(*
Nazwa:			FB_MoveRegister
Opis:			Blok przesuniecia rejestru formatek
Wersja:			v0.3 		
Data:			2018-11-16
Autor:			DP
Urzadzenia:		 
Konfiguracja:	
Info:
- Są dwa rejestry, wejściowy i wyjsciowy (struktury)
- Jezeli rejestr ma np. 6 elementów to za kazdym razem po wykryciu trigera program będzie
	1 wejściowy przesuwał na 1 wolny (nie ma formatki) wyjściowy
	kasował 1 rejestr wejściowy
	przesuwal rejetr wejsciowy 2 na 1(przeniesiony i skasowany), 3 na 2, 4 na 3, 5 na 4, 6 na 5 i kasowal 6wejsciowy
	tym sposobem po 6 trigerach caly rejestr wejsciowy powinien być na wyjsciowym
	np po 3 trigerach na wyjsciowym powinny byc zajete 1 do 3 i na wejsciowym 1 do 3
Błędy:
1 - nie wyszło z pętli for
2 - formatka już jest w rejestrze
Uwagi:
- 
Zmiany:
2018-09-18 Dodano sprawdzanie nasadek
2018-06-14 DP Pierwsza wersja
*)

FUNCTION_BLOCK FB_MoveRegisterLF
VAR_INPUT
	bFirstCycle:BOOL;					//Pierwszy cykl, zeby na początku nie wykrywało zbocza opadającego
	bTrigger :BOOL;						// Przesuniecie tablicy o jeden
	tTriggerFilterTimeOn:TIME:=T#0MS;	// Czas filtrowania wejścia Trigger na załączenie
	tTriggerFilterTimeOff:TIME:=T#0MS;	// Czas filtrowania wejścia Trigger na wyłączenie
	bTriggerBottle :BOOL;				// Zapisywanie czy jest butelka czy nie (jezeli kontrola wlączona)
	bWithBottleControl: BOOL;			// Włączona opcja kontroli butelek
	bWithCapControl:BOOL;				// Wlaczona kontrola nasadek
	bWithFormControlTrigerCounter:BOOL;	// Jezeku na trigercontrol nie ma formatki do przesunięcia to stwórz nową
	bMoveOnlyToLastExitRegister:BOOL;	// Przepisuj rejestr wejściowy tylko na ostatni wyjściowy bez przesunięcia wyjściowego
	bMoveOnlyIfFormPresent:BOOL;		// Przepisuj tylko jak jest formatka
	bRotateEntranceRegisterBefore:BOOL;	// Najpierw przesuń rejestr wejściowy a następnie z niego zabierz
	bNoKeepTryingMove:BOOL;				// Dalej przepisuj jezeli nie ma miejsca
	bTriggerCap: BOOL;					// Truger wykrycia nasadki
	bReset :BOOL;						// Czyszczenie tablic
	iEntranceArrayElements :UINT; 		// Wartość koncowa tablicy
	iExitArrayElements :UINT; 			// Wartość koncowa tablicy
	bInvertWriting :BOOL;				// Wpisywanie odwrotne zamist z 1entrance na 1exit to 1entrance na 6exit	
	eClearPackageState :S_PackageState; // Czysty rejestr
END_VAR
VAR_IN_OUT
	bTriggerCounter :BOOL;		// Triger ktory jest kasowany
	eEntranceState :ARRAY [1..17] OF S_PackageState;	
	eExitState :ARRAY [1..17] OF S_PackageState;
	bKeepTryingMove :BOOL;		// Probuj dalej zapisać formatki aż się któraś zwolni
END_VAR

VAR_OUTPUT	
	bError :BOOL; 				// Błąd
	iError: UINT;				// Nr Błędu
	bTriggerDone :BOOL; 		// Wykonano przesunięcie
	bTriggerFilteredOUT:BOOL;	//Wyjscie przefiltrowanego sygnalu wejsciowego
END_VAR

VAR
	i:UINT;						// Zmienna w tablicy
	k:UINT;						// Pomocnicza zmienna do zapisywnia czy jest butelka
	rtbTrigger :R_TRIG;			// Reaguje na zbocze
	rtbTriggerBottle :R_TRIG;	// Reaguje na zbocze
	rtbReset :R_TRIG;			// Reaguje na zbocze
	TimerResetErrors :TON;		// Reset Błedu
	nFormCounter :UINT;					//Licznik formatek
	r1,r2:UINT;
	bBottlePresent: BOOL;				//Zmienna pomocnicza ze wykryto butelkę
	bCapPresent: BOOL;					//Zmienna pomocnicza ze wykryto butelkę
	j: UINT;
	tonTriggerFilterTimeOn: TON;
	bTriggerFiltered: BOOL;
	tofTriggerFilterTimeOff: TOF;
	tonTriggerFilterTimeBeforeTrigger: TON;
END_VAR

//Filtrowanie sygnału wejściowego
tofTriggerFilterTimeOff	(IN:=bTrigger, PT:=tTriggerFilterTimeOff);
tonTriggerFilterTimeOn	(IN:=tofTriggerFilterTimeOff.Q, PT:=tTriggerFilterTimeOn);
bTriggerFiltered 		:= tonTriggerFilterTimeOn.Q;
bTriggerFilteredOUT		:= bTriggerFiltered ;

//TRIGI I TIMERY
IF bWithBottleControl THEN
	rtbTrigger 	(CLK := NOT bTriggerFiltered, Q=>);
	rtbTriggerBottle 	(CLK := NOT bTriggerBottle, Q=>);
ELSIF bWithCapControl THEN
	rtbTrigger 	(CLK := NOT bTriggerFiltered, Q=>);
ELSE
	rtbTrigger 	(CLK := bTriggerFiltered, Q=>);
	rtbTriggerBottle 	(CLK := bTriggerBottle, Q=>);
END_IF

rtbReset 	(CLK := bReset, Q=>);
TimerResetErrors (IN:= bError, PT:=T#1000MS, Q=>);

//RESETOWANIE BLEDU
IF TimerResetErrors.Q THEN
	bError := FALSE;
END_IF

//KASOWANIE ZMIENNYCH
bTriggerDone := FALSE;

//JEZELI WLACZONO KONTROLE BUTELEK TO NADPISUJ REJESTR CZY JEST BUTELKA
IF bWithBottleControl AND bTrigger AND bTriggerBottle AND NOT bKeepTryingMove THEN //Jezeli od wykrycia formatki liczy TIMER i wykryło butelke to wpisz do rejestru że jest butelka
	eEntranceState[1].bBottlePresent := TRUE;
	eEntranceState[1].bFormPresent := TRUE;
	bBottlePresent := TRUE; // Wpisuje że jest butelka jezeli wystąpi sygnał podczas trwania czujnika formatki
ELSIF bWithBottleControl AND rtbTrigger.Q AND NOT bBottlePresent AND  NOT bKeepTryingMove AND bFirstCycle THEN
	eEntranceState[1].bBottlePresent := FALSE;
	eEntranceState[1].bFormPresent := TRUE; // jeżeli zanik czujnik formatki i nie było formatki to wpisz ze nie było butelki
END_IF
//JEZELI WLACZONO KONTROLE NASADEk TO NADPISUJ REJESTR CZY JEST BUTELKA 
(*IF bWithCapControl AND bTrigger AND bTriggerCap AND NOT bKeepTryingMove THEN //Jezeli od wykrycia formatki liczy TIMER i wykryło butelke to wpisz do rejestru że jest butelka
	eEntranceState[1].bCapPutted := TRUE;
	eEntranceState[1].bCapOK := TRUE; eEntranceState[1].bBottlePresent:= TRUE;//Zmiana nowa
	eEntranceState[1].bFormPresent := TRUE;
	bCapPresent := TRUE; // Wpisuje że jest butelka jezeli wystąpi sygnał podczas trwania czujnika formatki*)
	//ZMIANA LU 192
IF bWithCapControl AND bTriggerCap AND NOT bKeepTryingMove THEN //Jezeli od wykrycia formatki liczy TIMER i wykryło butelke to wpisz do rejestru że jest butelka
	eEntranceState[1].bCapPutted := TRUE;
	eEntranceState[1].bCapOK := TRUE; eEntranceState[1].bBottlePresent:= TRUE;//Zmiana nowa
	eEntranceState[1].bFormPresent := TRUE;
	bCapPresent := TRUE; // Wpisuje że jest butelka jezeli wystąpi sygnał podczas trwania czujnika formatki	
ELSIF bWithCapControl AND rtbTrigger.Q AND NOT bCapPresent AND  NOT bKeepTryingMove AND bFirstCycle THEN
	eEntranceState[1].bCapPutted := TRUE;
	eEntranceState[1].bCapOK:= FALSE;
	eEntranceState[1].bFormPresent := TRUE; // jeżeli zanik czujnik formatki i nie było formatki to wpisz ze nie było butelki
END_IF
//JEZELI WLACZONO SPRAWDZANIE FORMATEK Z TRIGERCOUNTER TO
IF bWithFormControlTrigerCounter  AND (bTriggerCounter OR rtbTrigger.Q) AND NOT bKeepTryingMove AND bFirstCycle THEN //Zmiena UBL50, tworz tez nowa jak Trigger
	eEntranceState[1].bFormPresent := TRUE;
END_IF

IF rtbTrigger.Q OR bKeepTryingMove OR bTriggerCounter THEN
		bTriggerCounter := FALSE; 
		bKeepTryingMove := FALSE;
		nFormCounter := 0;
		bBottlePresent:= bCapPresent  := FALSE; 
		
			FOR j:=1 TO 3 DO
				FOR i:= 1 TO iExitArrayElements-1 DO // SORTOWANIE
					IF NOT eExitState[i].bFormPresent THEN 
						eExitState[i] := eExitState[i+1];
						eExitState[i+1] := eClearPackageState;
					END_IF
				END_FOR
			END_FOR	
		
			FOR i := 1 TO iEntranceArrayElements DO
				IF  NOT eExitState[i].bFormPresent THEN  		// Jeżeli w rejestrze wyjściowym jest wolne miejsce to wpisz rejestr wejściowy
					eExitState[i] := eEntranceState[1];	// Wpisz do rejestru dane np z [1] Buffor do [1,2,3,4,5,6] Package
					eEntranceState[1]:=eClearPackageState;	// Czyszczenie pierwszego rejestru wejściowego
					k:=i;											// Przepisywanie zmiennej pomocniczej
					FOR i := 1 TO iEntranceArrayElements DO   				
						IF i = iEntranceArrayElements THEN
							eEntranceState[i]:=eClearPackageState;		  // Zerowanie ostatniego bo zostało przesuniete wszystko o 1
						ELSE													  // Przepisanie 2 do 1, 3 do 2, 4 do 3, 5 do 4, 6 do 5, zeruj 6
							eEntranceState[i] := eEntranceState[i+1]; // 2 do 1, 3 do 2,
							eEntranceState[i+1]:=eClearPackageState;		  // zeruj 2, 
						END_IF
					END_FOR
					bTriggerDone := TRUE;
					EXIT;
					bError := TRUE;
					iError := 1;
				ELSE
					nFormCounter := nFormCounter + 1;
					bError := TRUE;
					iError := 2;
				END_IF
			END_FOR
		
		IF nFormCounter = iExitArrayElements THEN
		bKeepTryingMove:=NOT bNoKeepTryingMove;
		END_IF
	END_IF


//CZYSZCZENIE REJESTRU WEJSCIOWEGO
IF rtbReset.Q THEN
	FOR r1 := 1 TO iEntranceArrayElements DO
		eEntranceState[r1] := eClearPackageState;
	END_FOR
	FOR r2 := 1 TO iExitArrayElements DO
		eExitState[r2] := eClearPackageState;
	END_FOR
	bKeepTryingMove :=FALSE;
	bTriggerDone := FALSE;
	bTriggerCounter := FALSE; 
	nFormCounter := 0;
	bBottlePresent := bCapPresent := FALSE; 
	bError := FALSE;
	iError := 0;
END_IF

END_FUNCTION_BLOCK

(* stored: Version 1.1.0.1, ProductVersion 3.1.4026.13, FileIdentifier c59ff88f381e67ccd41827567cae2b57646bdfc1, FileSignature 57a3fbfcf8b111629a5d7783c2cdddf6111a52cc3706e7fa9ac359db5cdf741a17e6155f8b4dfe70d0a44c8dc2bf0f4ccbc864b478a3103516498a16e9a8371fa8479db2e1a0d90124ed975294b377b52c619078ca8a4b6239d16f891cedb55174ce8dc0df94b0e5068b0580f830ede2f2e3efd4be007abba6d94ee1e9c80f18bdac32d8376afec29250117908a5630c4d327a16521751376df453693292bf890d6f8eb689bf8bcafdffc77a765a22564ae5eec605e48478b49983b9514b01210803ae2f1a1192c5729e1a45c43458ab7f1de19ae0722b6de5e1318823431df3a986b29550af08dab9b65ec8dadb9dc53f2b5515b8622f860c728796913e2dbe
   POU FB_MoveRegisterLF: Id {4ce9c892-d077-4527-9ed4-05369faf27dd}, SpecialFunc None *)
